// TwinCAT 3 PLC project Coffee_Process
// ProgramVersion: 3.1.4024.0
// libraries:
//   Tc2_Standard, * (Beckhoff Automation GmbH)
//   Tc2_System, * (Beckhoff Automation GmbH)
//   Tc3_Module, * (Beckhoff Automation GmbH)
//   Util, * (System)
// project tree:
//   / Brewing.TcDUT, CoffeeMachine.TcDUT, GlobalTextList.TcGTLO, PlcTask.TcTTO, Visualization Manager.TcVMO (not stored)
//   GVLs/ GVL.TcGVL
//   POUs/ BrewCoffee.TcPOU, PrepareMachine.TcPOU, RefillWater.TcPOU
//   VISUs/ Process.TcVIS
// real-time tasks:
//   TASK PlcTask: cycle T#10ms, priority 1, ADS port 350

CONFIGURATION Coffee_Process
    RESOURCE PLC ON TwinCAT3
        TASK PlcTask(INTERVAL := T#10ms, PRIORITY := 20);
        PROGRAM BrewCoffee WITH PlcTask : BrewCoffee;
        PROGRAM PrepareMachine WITH PlcTask : PrepareMachine;
    END_RESOURCE
END_CONFIGURATION

// ---- Brewing.TcDUT
{attribute 'qualified_only'}
{attribute 'strict'}
TYPE Brewing :
(
	OFF,
	Idle,
	HeatingWater,
	BrewCoffee
):= OFF;
END_TYPE

// ---- CoffeeMachine.TcDUT
{attribute 'qualified_only'}
{attribute 'strict'}
TYPE CoffeeMachine :
(
	OFF,
	Standby,
	Waterfilled,
	PodPlaced,
	Ready
) := OFF;
END_TYPE

// ---- GVLs/GVL.TcGVL
{attribute 'qualified_only'}
VAR_GLOBAL
	Power				:		BOOL; // Turning On/Off the coffee machine
	StartBrewing		:		BOOL; //Preparing of machine is finished
	CoffeeBrewed		:		BOOL; // The coffee is brewed/finished
	WaterLevel			:		INT:= 4;
END_VAR

// ---- POUs/BrewCoffee.TcPOU
PROGRAM BrewCoffee
VAR
	WaterTemp			:		INT;
	LED					: 		BOOL;
	Timer				:		TON;

// STATES
	OFF					:		BOOL;			// Coffee machine is off
	Idle				:		BOOL;			// Waiting for input
	HeatingWater		:		BOOL;			// Water is heating up
   	BrewCoffee			: 		BOOL;			//
	State : Brewing := Brewing.OFF; 			// Current state
	
END_VAR

// Producing coffee by means of an senseo machine
// Name: Jurriën Arends
// Studentnumer: 515355
// Date: 21-10-2024
// Version: 0.6

// Task 2: Brewing coffee
CASE State OF	
// STATE OFF
Brewing.OFF:
     IF GVL.Power = FALSE THEN
	  OFF:= TRUE;
	  Idle:= FALSE;
	  LED:= FALSE;
    END_IF
	  
    IF GVL.Power = TRUE  THEN
	  State:= Brewing.Idle;
	  OFF:= FALSE;
    END_IF
	
  
 // STATE Idle 
 Brewing.Idle:
	IF GVL.Power = TRUE THEN
   	 Idle:= TRUE;
	 LED:= TRUE;
  	END_IF
	
	IF GVL.StartBrewing = TRUE THEN
		State:= Brewing.HeatingWater;
		WaterTemp:= 20;
		Idle:= FALSE;
		LED:= FALSE;
	END_IF
	
		IF GVL.Power = FALSE THEN
		state:= Brewing.OFF;
		LED:= OFF;
		Idle:= FALSE;
	END_IF
	

// State HeatingWater
Brewing.HeatingWater:
	IF GVL.StartBrewing = TRUE THEN
	 HeatingWater:= TRUE;
	 WaterTemp:= WaterTemp +1;
	 LED:= TRUE;
	 END_IF
	
	IF WaterTemp = 500 THEN
		state:= Brewing.BrewCoffee;
		HeatingWater:= FALSE;
		GVL.StartBrewing:= FALSE;
	END_IF
	
	IF GVL.Power = FALSE THEN
		state:= Brewing.OFF;
		LED:= OFF;
		HeatingWater:= FALSE;
	END_IF
	
// State BrewCoffee
Brewing.BrewCoffee:
	IF WaterTemp = 500 THEN
		BrewCoffee:= TRUE;
		LED:= TRUE;
	END_IF
	
	Timer(IN:=TRUE, PT:=T#5S);
	
	IF Timer.Q = TRUE THEN
		State:=Brewing.Idle;
		BrewCoffee:= FALSE;
		Timer(IN:= FALSE);
		GVL.CoffeeBrewed:= TRUE;
	END_IF
	
	IF GVL.Power = FALSE THEN
		state:= Brewing.OFF;
		LED:= OFF;
		BrewCoffee:= FALSE;
 	END_IF
	

ELSE
	OFF				:= TRUE;
	Idle			:= FALSE;
	HeatingWater	:= FALSE;
  	BrewCoffee		:= FALSE;
END_CASE;

END_PROGRAM

// ---- POUs/PrepareMachine.TcPOU
PROGRAM PrepareMachine
VAR
	LED					: 		BOOL;		// LED which indicates the machine is on/off or not enough water
	Pod					: 		BOOL;		// Pod(s) placed
	BlinkInterval		:		BLINK;		// Interval time for indicating there is not enough water
	CupsChoosen			:		BOOL;		// Amount of cups is choosen (1 or 2 cups)
	WaterRefilled		: 		BOOL;		// dddd
	
	// STATES
	OFF 				: 		BOOL;		// Coffee machine is off
	Standby 			:		BOOL;		// Coffee machine in standy mode
  	WaterFilled 		: 		BOOL;		// Water in machine needs to be filled
   	PodPlaced 			: 		BOOL;		// Pad(s) needs to be placed
	Ready				:		BOOL;		// Preparation is ready
	State : CoffeeMachine := CoffeeMachine.OFF; // Current state
	
	
END_VAR

// Producing coffee by means of an senseo machine
// Name: Jurriën Arends
// Studentnumer: 515355
// Date: 22-10-2024
// Version: 0.7

// The PLC program must contain:
// - 2 tasks running independently
// - 1 function called by at least one task 
// - a GVL from which the 2 tasks read and write variables


// Task 1: Preparing machine // DOWNLOAD LIBRARY BLINK
CASE State OF	
// STATE OFF
CoffeeMachine.OFF:
    IF GVL.Power = FALSE THEN
	  OFF:= TRUE;
	  Standby:= FALSE;
	  LED:= FALSE;
    END_IF
	
    IF GVL.Power = TRUE  THEN
	  State:= CoffeeMachine.Standby;
	  OFF:= FALSE;
    END_IF
	
	//IF WaterRefilled = TRUE THEN
	//	WaterLevel := 4;
	//	WaterRefilled:= FALSE;
	//END_IF
  
 // STATE Standby 
 CoffeeMachine.Standby:
  	IF GVL.Power = TRUE THEN
   	 Standby:= TRUE;
	 LED:= TRUE;
  	END_IF

	IF GVL.Power = FALSE  THEN
	  State:= CoffeeMachine.OFF;
	  Standby:= FALSE;
	  LED:= FALSE;
 	END_IF
	 
	IF GVL.WaterLevel <= 0  THEN
		BlinkInterval(ENABLE:= GVL.WaterLevel <=0, TIMELOW:= T#0.5S, TIMEHIGH:= T#0.5S, OUT=> LED);
		RefillWater(WaterRefilled);
		Waterrefilled:= FALSE;
		ELSIF GVL.WaterLevel > 0 THEN
		State:= CoffeeMachine.WaterFilled;
	 	Standby:= FALSE;
	  	LED:= FALSE;
	END_IF
	
	//IF WaterRefilled = TRUE THEN
	//	WaterLevel := 4;
	//	WaterRefilled:= FALSE;
	//END_IF
	
 // State WaterFilled 	
  CoffeeMachine.WaterFilled:
    IF GVL.WaterLevel > 0 THEN
      WaterFilled:= TRUE;
	  LED:= TRUE;
  	END_IF
	
 	IF Pod = TRUE THEN
	  State:= CoffeeMachine.PodPlaced;
	  WaterFilled:= FALSE;
	  LED:= FALSE;
  	END_IF
	
	IF GVL.Power = FALSE  THEN
	  State:= CoffeeMachine.OFF;
	  WaterFilled:= FALSE;
	  LED:= FALSE;
 	END_IF
	
	//IF WaterRefilled = TRUE THEN
	//	WaterLevel := 4;
	//	WaterRefilled:= FALSE;
	//END_IF
	 
	 	 
// State PodPlaced	
   CoffeeMachine.PodPlaced:
    IF Pod = TRUE THEN
      Podplaced:= TRUE;
	  LED:= TRUE;
 	END_IF
	
	IF CupsChoosen = TRUE THEN
	  State:= CoffeeMachine.Ready;
	  PodPlaced:= FALSE;
	  LED:= TRUE;
	END_IF
	
	 IF GVL.Power = FALSE  THEN
	  State:= CoffeeMachine.OFF;
	  PodPlaced:= FALSE;
	  LED:= FALSE;
 	 END_IF
	 
	 //IF WaterRefilled = TRUE THEN
	//	WaterLevel := 4;
	//	WaterRefilled:= FALSE;
	//END_IF
	 
// State Task ready	
   CoffeeMachine.Ready:
    IF CupsChoosen = TRUE THEN
      Ready:= TRUE;
	  LED:= TRUE;
	  GVL.StartBrewing:= TRUE;
	  Pod:= FALSE;
	  CupsChoosen:= FALSE;
 	END_IF
	
	 IF GVL.Power = FALSE  THEN
	  State:= CoffeeMachine.OFF;
	  Ready:= FALSE;
	  LED:= FALSE;
 	 END_IF
	 
	 IF GVL.CoffeeBrewed = TRUE THEN
		State:= CoffeeMachine.Standby;
		Ready:= FALSE;
		LED:= FALSE;
		GVL.WaterLevel := GVL.WaterLevel - 1;
		GVL.CoffeeBrewed:= FALSE;
	 END_IF
	 
	 IF Pod = TRUE THEN
      Pod:= FALSE;
	  LED:= TRUE;
 	END_IF
	 
	 //IF WaterRefilled = TRUE THEN
	//	WaterLevel := 4;
	//	WaterRefilled:= FALSE;
	//END_IF
ELSE
  OFF 			:= TRUE;
  Standby 		:= FALSE;
  WaterFilled 	:= FALSE;
  PodPlaced		:= FALSE;
  Ready			:= FALSE;
END_CASE;

END_PROGRAM

// ---- POUs/RefillWater.TcPOU
FUNCTION RefillWater : BOOL
VAR_INPUT
	WaterRefilled		:		BOOL;		// Water is refilled
END_VAR
VAR
END_VAR

// Refill water of coffee machine
IF WaterRefilled = TRUE THEN
  	GVL.WaterLevel := 2;
  	WaterRefilled:= FALSE;
END_IF;

END_FUNCTION

// ---- GlobalTextList.TcGTLO
TEXTLIST GlobalTextList
  16 = '/ WATERLEVEL'
  369 = 'BREW COFFEE STATE'
  845 = 'BREW COFFEE STATES'
  666 = 'BREWING'
  253 = 'Brewing Coffee'
  856 = 'CHOOSEN'
  391 = 'COFFEE'
  85 = 'CUPS'
  601 = 'Cups choosen'
  727 = 'FILLED'
  43 = 'HEATING'
  802 = 'Heating Water'
  334 = 'Idle'
  42 = 'IDLE'
  324 = 'INPUTS'
  3 = 'MACHINE'
  954 = 'Off'
  506 = 'OFF'
  816 = 'ON / OFF'
  515 = 'ON / OFF /'
  972 = 'On/Off/WaterLevel'
  987 = 'PadPlaced'
  596 = 'PLACED'
  212 = 'POD'
  955 = 'Pod Placed'
  158 = 'POWER'
  416 = 'Power '
  243 = 'Power On/Off'
  247 = 'Ready'
  562 = 'READY'
  143 = 'REFILL'
  928 = 'Refill Water'
  431 = 'Standby'
  272 = 'STANDBY'
  575 = 'STATE'
  702 = 'TASK: BREW COFFEE STATES'
  574 = 'TASK: PREPARE MACHINE STATES'
  898 = 'WATER'
  455 = 'Water Filled'
  184 = 'WaterFilled'
  456 = 'WATERLEVEL'
END_TEXTLIST

// ---- VISUs/Process.TcVIS
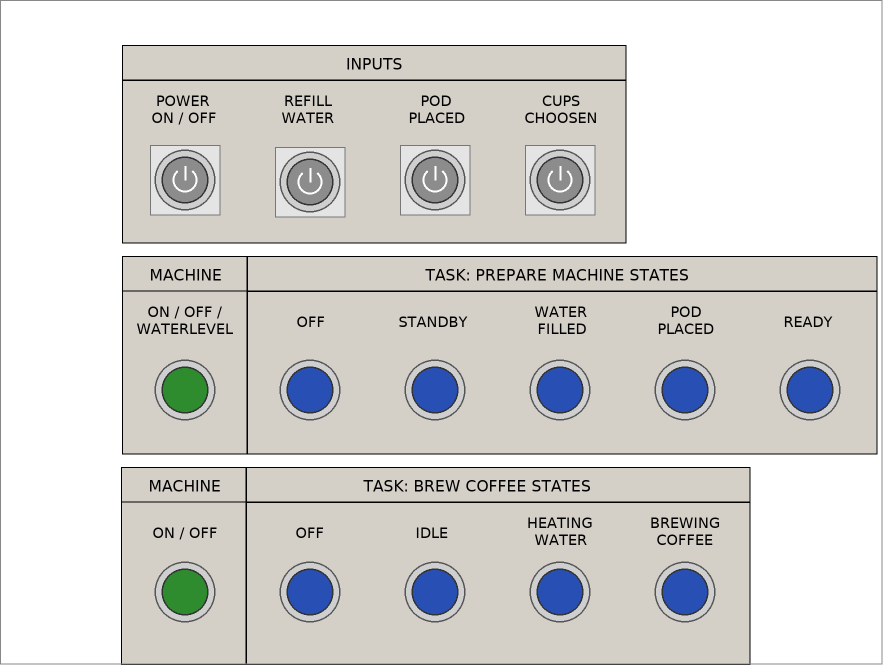
VISUALIZATION Process  // 883x665
    Rectangle (247,291 630x163)
    Rectangle (247,256 630x35)
    Rectangle (122,256 125x198)
    Label (358,307 150x30), "STANDBY"
    Label (236,307 150x30), "OFF"
    Label (486,297 150x30), "WATER"
    Label (611,297 150x30), "POD"
    Rectangle (122,256 125x35)
    Label (111,260 150x30), "MACHINE"
    Label (487,314 150x30), "FILLED"
    Label (611,314 150x30), "PLACED"
    Label (395,260 325x30), "TASK: PREPARE MACHINE STATES"
    Rectangle (246,502 504x163)
    Rectangle (246,467 504x35)
    Rectangle (121,467 125x198)
    Lamp1 (150,355 70x70), variable: PrepareMachine.LED, style: Lamp-Lamp1-Green
    Lamp1 (275,355 70x70), variable: PrepareMachine.OFF, style: Lamp-Lamp1-Blue
    Lamp1 (400,355 70x70), variable: PrepareMachine.Standby, style: Lamp-Lamp1-Blue
    Lamp1 (525,355 70x70), variable: PrepareMachine.WaterFilled, style: Lamp-Lamp1-Blue
    Lamp1 (650,355 70x70), variable: PrepareMachine.PodPlaced, style: Lamp-Lamp1-Blue
    Lamp1 (775,355 70x70), variable: PrepareMachine.Ready, style: Lamp-Lamp1-Blue
    Label (110,518 150x30), "ON / OFF"
    Label (357,518 150x30), "IDLE"
    Label (235,518 150x30), "OFF"
    Label (485,508 150x30), "HEATING"
    Label (610,508 150x30), "BREWING"
    Lamp1 (650,557 70x70), variable: BrewCoffee.BrewCoffee, style: Lamp-Lamp1-Blue
    Lamp1 (525,557 70x70), variable: BrewCoffee.HeatingWater, style: Lamp-Lamp1-Blue
    Lamp1 (400,557 70x70), variable: BrewCoffee.Idle, style: Lamp-Lamp1-Blue
    Lamp1 (275,557 70x70), variable: BrewCoffee.OFF, style: Lamp-Lamp1-Blue
    Lamp1 (150,557 70x70), variable: BrewCoffee.LED, style: Lamp-Lamp1-Green
    Rectangle (121,467 125x35)
    Label (110,471 150x30), "MACHINE"
    Label (486,525 150x30), "WATER"
    Label (610,525 150x30), "COFFEE"
    Label (347,471 261x30), "TASK: BREW COFFEE STATES"
    Label (110,297 150x30), "ON / OFF /"
    Label (110,314 150x30), "WATERLEVEL"
    Label (733,307 150x30), "READY"
    Rectangle (122,80 504x163)
    Rectangle (122,45 504x35)
    Label (361,86 150x30), "POD"
    Label (486,86 150x30), "CUPS"
    Label (362,103 150x30), "PLACED"
    Label (486,103 150x30), "CHOOSEN"
    Label (244,49 261x30), "INPUTS"
    Label (108,86 150x30), "POWER"
    Label (233,86 150x30), "REFILL"
    Label (109,103 150x30), "ON / OFF"
    Label (233,103 150x30), "WATER"
    PowerSwitch (150,145 70x70), variable: GVL.Power, behaviour: TOGGLE, style: Switch-PowerSwitch-Gray
    PowerSwitch (400,145 70x70), variable: PrepareMachine.Pod, behaviour: TOGGLE, style: Switch-PowerSwitch-Gray
    PowerSwitch (525,145 70x70), variable: PrepareMachine.CupsChoosen, behaviour: TOGGLE, style: Switch-PowerSwitch-Gray
    PowerSwitch (275,147 70x70), variable: PrepareMachine.WaterRefilled, behaviour: TOGGLE, style: Switch-PowerSwitch-Gray
END_VISUALIZATION
